Staubli VAL3: insertInstr.pgx

program insertInstr()
  local num i
  local string l_sMessage
  local num l_nIndex
  local string l_sItem
  local string l_sPath
begin
//  // create the list
//  call use:setSizeList(19,0,19,11)
//  call use:setView(false)
//  call language:message(l_sMessage,35)
//  call use:listcreate(l_sMessage)
//  // insert the action on Point
//  call use:listadd(saveData:sInstrOnPoint)
//  call use:listupdate(0)
//  // SELECT THE ITEM
//  x_iInstr.sData=""
//  do
//    i=get()
//    l_nIndex=0
//    call use:listevent(i,l_nIndex,l_sItem)
//  until i==255 or i==270
//  // update
//  x_iInstr.sType=l_sItem
//  // update
//  call saveData:getPathInstr(l_sItem,l_sPath)
//  if l_sItem!="" and i==270
//    events:libLoad(l_sPath)
//    delay(0)
//    call events:onInsert(l_sItem)
//    x_iInstr.sData=l_sItem
//  endIf
end
